ABB RAPID module: main.rapid

MODULE main
  ! RAPID Tool - Kinematic Solver
  ! Objective: Deterministic kinematic solver for articulated robotic manipulators

  ! Define world object
  VAR robtarget pHome;!

  ! Define robot tool and workobject
  VAR tooldata tWelding;!
  VAR wobjdata wPart;!

  ! Main procedure
  PROC main()
    ! Initialize home position
    pHome.x:= 500;
    pHome.y:= -200;
    pHome.z:= 400;
    pHome.qpos1:= 0;
    pHome.qpos2:= 0;
    pHome.qpos3:= 0;
    pHome.qpos4:= 0;

    ! Move to home position
    MoveJ pHome, v1000, z50, tWelding;

    ! Perform kinematic calculation (placeholder)
    ! This would typically involve inverse kinematics calculations
    ! based on desired end-effector pose

    ! Example movement to a calculated point
    VAR robtarget pTarget;!
    pTarget.x:= 600;
    pTarget.y:= 0;
    pTarget.z:= 300;
    pTarget.qpos1:= 0.707;
    pTarget.qpos2:= 0;
    pTarget.qpos3:= 0;
    pTarget.qpos4:= -0.707;

    MoveL pTarget, v100, z50, tWelding;

    ! Return to home
    MoveJ pHome, v1000, z50, tWelding;
  ENDPROC

ENDMODULE
